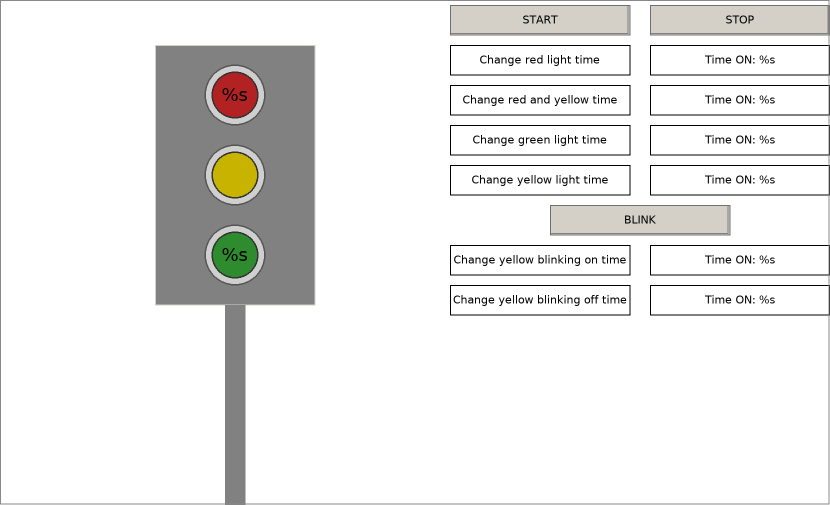
VISUALIZATION Visualization  // 830x505
    Rectangle (155,45 160x260)
    Lamp1 (200,60 70x70), variable: MAIN.fbTrafficLight.bTurnRedLightOn, style: Lamp-Lamp1-Red
    Lamp1 (200,140 70x70), variable: MAIN.fbTrafficLight.bTurnYellowLightOn, style: Lamp-Lamp1-Yellow
    Lamp1 (200,220 70x70), variable: MAIN.fbTrafficLight.bTurnGreenLightOn, style: Lamp-Lamp1-Green
    Rectangle (225,305 20x200)
    Rectangle (450,45 180x30), "Change red light time"
        OnMouseClick: write MAIN.dwRedTimeOn via Default
    Rectangle (450,85 180x30), "Change red and yellow time"
        OnMouseClick: write MAIN.dwRedAndYellowTimeOn via Default
    Rectangle (450,125 180x30), "Change green light time"
        OnMouseClick: write MAIN.dwGreenTimeOn via Default
    Rectangle (450,165 180x30), "Change yellow light time"
        OnMouseClick: write MAIN.dwYellowTimeOn via Default
    Rectangle (220,80 30x30), "%s", text variable: MAIN.fbTrafficLight.dwRedTimeRemaining, invisible if: NOT MAIN.fbTrafficLight.bTurnRedLightOn OR MAIN.fbTrafficLight.bTurnYellowLightOn
    Rectangle (220,240 30x30), "%s", text variable: MAIN.fbTrafficLight.dwGreenTimeRemaining, invisible if: NOT (MAIN.fbTrafficLight.eLightOrder = 300)
    Rectangle (450,245 180x30), "Change yellow blinking on time"
        OnMouseClick: write MAIN.dwYellowBlinkingTimeOn via Default
    Rectangle (450,285 180x30), "Change yellow blinking off time"
        OnMouseClick: write MAIN.dwYellowBlinkingTimeOff via Default
    Rectangle (650,45 180x30), "Time ON: %s", text variable: MAIN.fbTrafficLight.fbRedTimerOn.ET
    Rectangle (650,85 180x30), "Time ON: %s", text variable: MAIN.fbTrafficLight.fbRedAndYellowTimerOn.ET
    Rectangle (650,125 180x30), "Time ON: %s", text variable: MAIN.fbTrafficLight.fbGreenTimerOn.ET
    Rectangle (650,165 180x30), "Time ON: %s", text variable: MAIN.fbTrafficLight.fbYellowTimerOn.ET
    Rectangle (650,245 180x30), "Time ON: %s", text variable: MAIN.fbTrafficLight.fbYellowBlinker.fbTimerOn.ET
    Rectangle (650,285 180x30), "Time ON: %s", text variable: MAIN.fbTrafficLight.fbYellowBlinker.fbTimerOff.ET
    Button (450,5 180x30), "START"
        tap MAIN.bIsStartPressed
    Button (650,5 180x30), "STOP"
        tap MAIN.bIsStopPressed
    Button (550,205 180x30), "BLINK"
        tap main.bIsBlinkPressed
END_VISUALIZATION

(* stored: Version 1.1.0.1, ProductVersion 3.1.4024.12
   Visu Visualization: Id {34d7f575-93eb-4ab0-9a60-0d4a07b45ad2} *)
